FUNCTION_BLOCK Queue EXTENDS FB_BaseFb
VAR_INPUT
	{attribute 'OPC.UA.DA' := '0'}
	busySem : BOOL :=FALSE; //used for test and set from outside call
END_VAR

VAR_OUTPUT
	
END_VAR
{attribute 'OPC.UA.DA' := '0'}
VAR CONSTANT
     QUEUE_SIZE  : UINT := 15;
END_VAR

VAR
	{attribute 'OPC.UA.DA' := '0'}
	StructSize : UDINT;
	{attribute 'OPC.UA.DA' := '0'}
	QArr	: ARRAY[0..QUEUE_SIZE] OF STRING[1000];	
	{attribute 'OPC.UA.DA' := '0'}
	pQArr  : POINTER TO  STRING;	
	{attribute 'OPC.UA.DA' := '0'}
	QWriteAdr :POINTER TO  STRING;
	{attribute 'OPC.UA.DA' := '0'}
	QReadAdr : POINTER TO  STRING;
	{attribute 'OPC.UA.DA' := '0'}
	pRead : UDINT;
	{attribute 'OPC.UA.DA' := '0'}
	pWrite :UDINT;
	{attribute 'OPC.UA.DA' := '0'}
	isInitDone :BOOL;
	{attribute 'OPC.UA.DA' := '0'}
	IsOverflow : BOOL;
	{attribute 'OPC.UA.DA' := '0'}
	isBusy :BOOL;	
	{attribute 'OPC.UA.DA' := '0'}
	isFull	: BOOL;
	{attribute 'OPC.UA.DA' := '0'}
	o_isEmpty : BOOL;
	{attribute 'OPC.UA.DA' := '0'}
	Error : BOOL;
	{attribute 'OPC.UA.DA' := '0'}
	ErrorID :USINT;
	{attribute 'OPC.UA.DA' := '0'}
	WriteMsgCount : UDINT;
	{attribute 'OPC.UA.DA' := '0'}
	ReadMsgCount  : UDINT;
	{attribute 'OPC.UA.DA' := '0'}
	o_EntriesCount : UINT;
	
END_VAR

METHOD CheckQReadAvailable : BOOL
VAR_INPUT
END_VAR

IF (isEmpty=FALSE) AND (isBusy = FALSE) THEN
	CheckQReadAvailable:= TRUE;
ELSE	
	CheckQReadAvailable:= FALSE;	
END_IF
END_METHOD

METHOD CheckQWriteAvailable : BOOL
VAR_INPUT
END_VAR

IF (isFull=FALSE) AND (isBusy = FALSE) THEN
	CheckQWriteAvailable:= TRUE;
	
ELSE
	
	CheckQWriteAvailable:= FALSE;	
END_IF
END_METHOD

METHOD Clear : BOOL
VAR_INPUT
END_VAR
		memset(pQArr,0,SIZEOF(QArr));
		pRead		:=0;
		pWrite		:=0;
		
		isInitDone 		:= TRUE;
		o_isEmpty		:=TRUE;
		isFull			:=FALSE;	
		isBusy			:=FALSE;
		Error			:=FALSE;
		ErrorID			:=0;
		
		o_EntriesCount := 0;
END_METHOD

METHOD Dequeue : BOOL
VAR_INPUT
	pReadData : POINTER TO BYTE;
	MsgLength  : UDINT;
END_VAR

IF THIS^.o_EntriesCount > 0 THEN	
	QReadAdr		:= (pQArr)+(pRead*StructSize);	
	memcpy(pReadData,QReadAdr,MsgLength);// (pDest,pSrc,length)
	THIS^.o_EntriesCount	:= THIS^.o_EntriesCount - 1;	
	pRead:=pRead+1;
	
	IF THIS^.pRead >= QUEUE_SIZE THEN
		THIS^.pRead	:= 0;
	END_IF	
	
    THIS^.IsFull		:= FALSE;
	ReadMsgCount:=ReadMsgCount+1;
	IF pRead=pWrite THEN
		o_isEmpty:=TRUE;
	END_IF	
		
END_IF
END_METHOD

METHOD Enqueue : BOOL
VAR_INPUT
	pWriteData : POINTER TO BYTE;	
	MsgLength  : UDINT;
END_VAR
IF o_EntriesCount < QUEUE_SIZE THEN
	isBusy := TRUE;
	QWriteAdr				:=(pQArr)+(pWrite*StructSize);
		IF MsgLength>0 AND (MsgLength<=StructSize)THEN
			memcpy(QWriteAdr,pWriteData,MsgLength);// (pDest,pSrc,length)  		
		ELSIF (MsgLength>StructSize)THEN
			Error		:=TRUE;
			ErrorID 	:= 5;
			memcpy(QWriteAdr,pWriteData,StructSize);// (pDest,pSrc,length)
		ELSE	// MsgLength = 0
			memcpy(QWriteAdr,pWriteData,StructSize);// (pDest,pSrc,length)	
		END_IF;
		pWrite:=pWrite+1;
		WriteMsgCount:=WriteMsgCount+1;
	// increase entries counter
	THIS^.o_EntriesCount	:= THIS^.o_EntriesCount + 1;	
		
	IF pWrite>=(QUEUE_SIZE) THEN
		pWrite:=0;
	END_IF;	
	
	THIS^.o_isEmpty		:= FALSE;
	IF THIS^.o_EntriesCount >= QUEUE_SIZE THEN
		THIS^.IsFull	:= TRUE;
	END_IF	
	
	IF WriteMsgCount>10000000 THEN
		WriteMsgCount:=0;
	END_IF;			
	isBusy := FALSE;
ELSE
	THIS^.IsOverflow	:= TRUE;	
END_IF
END_METHOD

PROPERTY EntriesCount : UINT
GET
EntriesCount :=o_EntriesCount;
END_GET
SET
END_SET
END_PROPERTY

METHOD FB_init : BOOL
VAR_INPUT
	bInitRetains : BOOL; // if TRUE, the retain variables are initialized (warm start / cold start)
	bInCopyCode : BOOL;  // if TRUE, the instance afterwards gets moved into the copy code (online change)
END_VAR
		THIS^.pQArr := ADR(QArr);		
		StructSize := SIZEOF(QArr[0]);
		
		memset(pQArr,0,SIZEOF(QArr));
		pRead		:=0;
		pWrite		:=0;
		
		isInitDone 		:= TRUE;
		o_isEmpty		:=TRUE;
		isFull			:=FALSE;	
		isBusy			:=FALSE;
		Error			:=FALSE;
		ErrorID			:=0;
		
		o_EntriesCount := 0;
END_METHOD

PROPERTY isEmpty : BOOL
GET
isEmpty := o_isEmpty;
END_GET
SET
END_SET
END_PROPERTY

METHOD Peek : BOOL
VAR_INPUT
END_VAR
END_METHOD

METHOD ReadCurrentEntry : BOOL//Only Read not Pop
VAR_INPUT
	pReadData : POINTER TO BYTE;
	MsgLength  : UDINT;
END_VAR

IF THIS^.o_EntriesCount > 0 THEN	
	QReadAdr		:= (pQArr)+(pRead*StructSize);	
	memcpy(pReadData,QReadAdr,MsgLength);// (pDest,pSrc,length)
	ReadCurrentEntry := TRUE;	
ELSE
	ReadCurrentEntry := FALSE;	
END_IF
END_METHOD

END_FUNCTION_BLOCK

(* stored: Version 1.1.0.1, ProductVersion 3.1.4024.3
   POU Queue: Id {9a463fdc-e8d3-07a5-2df7-6a5578f8093e}, SpecialFunc None
   Method CheckQReadAvailable: Id {2a650440-47e4-0d42-246b-cd27ce1cc385}
   Method CheckQWriteAvailable: Id {ce7ed7ce-c16d-0097-03f7-acc174f675f3}
   Method Clear: Id {7970bdfd-2714-069e-3b2a-195de24d219c}
   Method Dequeue: Id {f3e3a0a4-efd7-087d-1ffd-d76f020ca27a}
   Method Enqueue: Id {8a114534-2d18-0753-2333-1da3bd1e71bd}
   Property EntriesCount: Id {db997301-0655-0fea-2a92-0a5b756acc2a}
   Get Get: Id {bb9369b1-93d4-0c3e-152e-fa5eab18c4a2}
   Set Set: Id {15be1695-e071-0913-1985-a9298d2f096c}
   Method FB_init: Id {aa37b90b-1ec2-0d2d-034c-ac8d42c24842}
   Property isEmpty: Id {2f202cc8-4cb0-0ff3-1044-88a7ce651056}
   Get Get: Id {4c18bd07-2589-0f62-2987-42d5c2848ac8}
   Set Set: Id {51a20d30-5e8e-0701-1b69-c08e2c5db79e}
   Method Peek: Id {6c157c0d-dff1-0582-27db-323ce1b00d25}
   Method ReadCurrentEntry: Id {9f36baeb-fc72-09c4-2e61-62a1aca635d6} *)
